// TIA Portal V19 export
TYPE "Positioning_MOL_Machine_Config"
// stored: Access Published
   STRUCT
      DelayMissingCondition : Time;
      CyclicOBTime_ms : LReal;
      Ax : "OOAx_Config";
      Ax_UM2 : "udt_LinTranformation";
   END_STRUCT;
END_TYPE
